FUNCTION_BLOCK PUBLIC FB_MyFoo EXTENDS MyNamespace01.FB_Foo IMPLEMENTS MyNamespace01.I_Foo
VAR_INPUT
END_VAR
VAR_OUTPUT
END_VAR
VAR
END_VAR

{warning 'add method implementation'}
METHOD DoSomething : BOOL
END_METHOD

END_FUNCTION_BLOCK

(* stored: Version 1.1.0.1, ProductVersion 3.1.4020.6
   POU FB_MyFoo: Id {dfa4b2f9-375e-485b-b1c1-6e3405e8ec5f}, SpecialFunc None
   Method DoSomething: Id {b75fdda0-0d73-4019-abcd-e4a1b86e5430} *)
